PROGRAM MAIN
VAR
	AdsRead:						ADSREADEX;
	ADSReadWrite:					ADSRDWRT;
	SymbolUploadInfo:				TAdsSymbolUploadInfo;
	DestBuffer:						ARRAY [0..100] OF BYTE;
	SrcBuffer:						STRING;
	pTypeInfo:						POINTER TO BYTE;
	ReadSymbolTableState:			TReadSymbolTableState;
	ReadSymbolTableStatePrev:		TReadSymbolTableState;
	start:							BOOL;
	pAdsDatatypeEntry:				POINTER TO AdsSymbolEntry;
	pSubAdsDatatypeEntry:			POINTER TO AdsSymbolEntry;
	pNameStringPointer:				POINTER TO STRING;
	pTypeStringPointer:				POINTER TO STRING;
	NameString:						STRING;
	TypeString:						STRING;
	pSubNameStringPointer:			POINTER TO STRING;
	SubNameString:					STRING;
	iterate:						BOOL;
	i:								UDINT;

END_VAR

CASE ReadSymbolTableState OF
	RS_WAIT_FOR_START:
		IF(start = TRUE)THEN 	
			start := FALSE;
			AdsRead(
				PORT := 851, 
				DESTADDR := ADR(SymbolUploadInfo),
				IDXGRP := 16#F00C,
				IDXOFFS := 0,
				LEN := SIZEOF(SymbolUploadInfo),
				READ := TRUE
					);
			ReadSymbolTableState := RS_READ_SYMBOL_UPLOAD_INFO;
		END_IF
		
	RS_READ_SYMBOL_UPLOAD_INFO:	
		AdsRead();
		IF(AdsRead.BUSY = FALSE)THEN
			AdsRead(Read := FALSE);
			pTypeInfo := __NEW(BYTE, SymbolUploadInfo.nSymSize);			
			ReadSymbolTableState := RS_READ_SYMBOL_UPLOAD_START;	
		END_IF	
		
	RS_READ_SYMBOL_UPLOAD_START:
		AdsRead();
		IF(AdsRead.BUSY = FALSE)THEN
			AdsRead(
				PORT := 851, 
				DESTADDR := pTypeInfo,
				IDXGRP := 16#F00B,
				IDXOFFS := 0,
				LEN := SymbolUploadInfo.nSymSize,
				READ := TRUE
					);
			ReadSymbolTableState := RS_READ_SYMBOL_UPLOAD;
		END_IF
		
	RS_READ_SYMBOL_UPLOAD: 		
	
		AdsRead();
		IF(AdsRead.BUSY = FALSE)THEN
			pAdsDatatypeEntry := pTypeInfo;
			i := 0;
			ReadSymbolTableState := RS_PROCESS_SYMBOL_UPLOAD;		
		END_IF
			
	RS_PROCESS_SYMBOL_UPLOAD:
		IF(i< SymbolUploadInfo.nSymbols-1)THEN
			pNameStringPointer := pAdsDatatypeEntry + 30 (* Sizeof(AdsDatatypeEntry) geeft net wat teveel*);
			NameString := pNameStringPointer^;
			LogMsg(NameString);
			
 			pTypeStringPointer := + pNameStringPointer + pAdsDatatypeEntry^.nameLength + 1;
			TypeString := pTypeStringPointer^;
			LogMsg(TypeString);
(*			IF(pAdsDatatypeEntry^.subItems > 0)THEN
				//Sub item:
				pSubAdsDatatypeEntry := pNameStringPointer + pAdsDatatypeEntry^.nameLength+1 + pAdsDatatypeEntry^.typeLength+1 + pAdsDatatypeEntry^.commentLength+1 + 8; 
				pSubNameStringPointer := pSubAdsDatatypeEntry + 42 (* Sizeof(AdsDatatypeEntry) geeft net wat teveel*);
				SubNameString := pSubNameStringPointer^;
				TracePrintString(SubNameString);
			END_IF*)			
			pAdsDatatypeEntry := pAdsDatatypeEntry + pAdsDatatypeEntry^.entryLength;
			i := i + 1;
		ELSE
			ReadSymbolTableState := RS_DONE;
		END_IF
		
		
	RS_DONE:
		;		

100:
	ADSReadWrite(
		PORT := 851,
		SRCADDR :=  ADR(SrcBuffer),
		DESTADDR := ADR(DestBuffer)
			);
END_CASE
(*
CASE ReadSymbolTableState OF
	0:
		IF(start = TRUE)THEN 	
			start := FALSE;
			AdsRead(
				PORT := 851, 
				DESTADDR := ADR(SymbolUploadInfo),
				IDXGRP := 16#F00F,
				IDXOFFS := 0,
				LEN := SIZEOF(SymbolUploadInfo),
				READ := TRUE
					);
			ReadSymbolTableState := 1;
		END_IF
		
	1:	
		AdsRead();
		IF(AdsRead.BUSY = FALSE)THEN
			AdsRead(Read := FALSE);
			pTypeInfo := __NEW(BYTE, SymbolUploadInfo.nDatatypeSize);			
			ReadSymbolTableState := 2;	
		END_IF	
		
	2:
		AdsRead();
		IF(AdsRead.BUSY = FALSE)THEN
			AdsRead(
				PORT := 851, 
				DESTADDR := pTypeInfo,
				IDXGRP := 16#F00E,
				IDXOFFS := 0,
				LEN := SymbolUploadInfo.nDatatypeSize,
				READ := TRUE
					);
			ReadSymbolTableState := 3;
		END_IF
		
	3: 		
		AdsRead();
		IF(AdsRead.BUSY = FALSE)THEN
			pAdsDatatypeEntry := pTypeInfo;
			ReadSymbolTableState := 4;
		END_IF
			
	4:
		FOR i := 0 TO SymbolUploadInfo.nDatatypes DO
					
			pNameStringPointer := pAdsDatatypeEntry + 42 (* Sizeof(AdsDatatypeEntry) geeft net wat teveel*);
			NameString := pNameStringPointer^;
			TracePrintString(NameString);
			IF(NameString = 'TSymbolUploadInfo')THEN
				iterate := FALSE;	
			END_IF
			IF(pAdsDatatypeEntry^.subItems > 0)THEN
				//Sub item:
				pSubAdsDatatypeEntry := pNameStringPointer + pAdsDatatypeEntry^.nameLength+1 + pAdsDatatypeEntry^.typeLength+1 + pAdsDatatypeEntry^.commentLength+1 + 8; 
				pSubNameStringPointer := pSubAdsDatatypeEntry + 42 (* Sizeof(AdsDatatypeEntry) geeft net wat teveel*);
				SubNameString := pSubNameStringPointer^;
				TracePrintString(SubNameString);
			END_IF			
			pAdsDatatypeEntry := pAdsDatatypeEntry + pAdsDatatypeEntry^.entryLength;
		END_FOR
		ReadSymbolTableState := 5;
		
		

100:
	ADSReadWrite(
		PORT := 851,
		SRCADDR :=  ADR(SrcBuffer),
		DESTADDR := ADR(DestBuffer)
			);
END_CASE

*)

LogStateChange();
ReadSymbolTableStatePrev := ReadSymbolTableState;

gTime := gTime + 1;

METHOD LogStateChange : BOOL
VAR_INPUT
END_VAR
IF(ReadSymbolTableState <> ReadSymbolTableStatePrev)THEN
	LogMsg(concat(concat(TO_STRING(ReadSymbolTableStatePrev), ' => '), TO_STRING(ReadSymbolTableState)));
END_IF
END_METHOD

END_PROGRAM

(* stored: Version 1.1.0.1, ProductVersion 3.1.4024.3
   POU MAIN: Id {749b57ec-766c-486f-8c5f-78c0399fac58}, SpecialFunc None
   Method LogStateChange: Id {3e911aee-3a56-48b2-acf3-e97822254fc6} *)
